TYPE UNIFIED_PROGRAM_STEP_ACTION :
STRUCT
	Name : STRING;
	Args : ARRAY [0..UnifiedProgramConstants.MaxActionArgumentsCount - 1] OF STRING(255);
END_STRUCT
END_TYPE

(* stored: Version 1.1.0.1
   DUT UNIFIED_PROGRAM_STEP_ACTION: Id {f92efd89-ea51-4d53-86a8-2706751d7804} *)
